{attribute 'qualified_only'}
{attribute 'strict'}
TYPE eOB_StopBeforeVisionState :
( 
	eUnknown,
    eInit,
	eHoming,
	eReady,
	eDwell,
	eProcessing,
	eDepart,
	eStopActive,
    eError
);
END_TYPE

(* stored: Version 1.1.0.1, ProductVersion 3.1.4020.12
   DUT eOB_StopBeforeVisionState: Id {95274ef1-8b64-4c31-923f-dd9c11cf0c65} *)
